// TIA Portal V18 export
TYPE "TANK DATA"
// stored: IsFailsafeCompliant false
   STRUCT
      "TANK TEMP SP" : Real;
      "LINE TEMP SP" : Real;
      "RETURN SP" : Real;
      "COND SP" : Real;
      "HYSTERIRIS TEMP" : Real;
      "HYSTERISIS COND" : Real;
      "CYCLE TIME MIN" : Int;
      "CYCLE TIME SEC" : Int;
      "ELAPSED MIN" : Int;
      "ELAPSED SEC" : Int;
   END_STRUCT;
END_TYPE
